FUNCTION_BLOCK Alarms_FB EXTENDS FB_TcAlarm
VAR_INPUT
	evtEntry : TcEventEntry;
	bEvt : BOOL;
	bConfirm : BOOL;
END_VAR
VAR_OUTPUT
END_VAR
VAR
	bInit  : BOOL := TRUE;
	bMem : BOOL;
END_VAR

IF bInit THEN
	SUPER^.CreateEx(evtEntry, TRUE, 0);
	bInit := FALSE;
END_IF

IF bEvt AND NOT bMem AND SUPER^.eConfirmationState <> TcEventConfirmationState.WaitForConfirmation THEN
	SUPER^.Raise(0);
END_IF

IF bMem AND NOT bEvt THEN
	SUPER^.Clear(0, FALSE);
END_IF

IF bConfirm THEN
	SUPER^.Confirm(0);
END_IF
bMem := bEvt;

END_FUNCTION_BLOCK

(* stored: Version 1.1.0.1, ProductVersion 3.1.4024.11
   POU Alarms_FB: Id {52c4c7da-671c-4ba9-a4b5-2dc31bdbccec}, SpecialFunc None *)
